INTERFACE I_PMLSubUnitInfo EXTENDS I_InterfaceBase

END_INTERFACE

(* stored: Version 1.1.0.1, ProductVersion 3.1.4024.12
   Itf I_PMLSubUnitInfo: Id {b4b37584-2e9c-4c24-ba11-c9388eeb6837} *)
